FUNCTION "TestOnceMore" : Void
{ S7_Optimized_Access := 'TRUE' }
VERSION : 0.1
   VAR_INPUT
      A : Bool;
   END_VAR

   VAR_OUTPUT
      B : Bool;
   END_VAR


BEGIN

	#B := #A;

END_FUNCTION

